# B&R Automation Studio project PLC
Automation Studio 4.7.2.98

## Configuration Config1

CPU X20CP1586, AutomationRuntime C4.72, Build 4.1.2, Vc V4.72.0

### Task classes (Cpu.sw)
```
Cyclic#4:
  Program <- Program.prg
```

### Hardware
```
X20CP1586 : X20CP1586 v1.6.0.0
```

## Logical view

### Program Logical/Program

#### Main.st
```iecst
PROGRAM _INIT
	(* Insert code here *)

END_PROGRAM

PROGRAM _CYCLIC
	(* Insert code here *)
	(*Ready*)

END_PROGRAM

PROGRAM _EXIT
	(* Insert code here *)

END_PROGRAM
```
